(* IEC 61131-3 sources: Dev/Dev_V200/200 (part 23) *)

VAR_GLOBAL
	fb_Nh_Create_DIR		: _Nh_Create_DIR;
END_VAR

{ $DEFINE __NH_LIST_PLC_STRING }

TYPE
   NH_FRM_HED {HIDDEN}   : STRUCT      				// HLAVNA RIADIACA PREMENNA
      name     : STRING[5] :='_END';
		desc		: STRING[20];
      wht      : USINT;       	// 1-brw,2-FRM,3-MNU,4- HOME-PG - ALL, 0=read All file (log/230...)
		row		: USINT:=1;       // numbrer of Rows
		sld		: USINT;    		// number of sliders
		siz		: UDINT;				// size all file (NH_FRM_HED+data)
	END_STRUCT;

	NH_PLC_DIR_DHED       : STRUCT   	// dir
//      eTime   	: STRING[11] :='00:00:00.00'; stim 	: BYTE := 16#3b;
      dUp   	: STRING[1] :=' ';
		dEmpty	: STRING[1]	:=' ';
      dDT   	: STRING[19]:='                   ';
//		dName		: STRING;	//:='                                                                           ';
//      Cr       : BYTE   := 16#0D;
//      Lf       : BYTE   := 16#0A;
	END_STRUCT;
	{ $IFDEF __NH_LIST_PLC_STRING }
		NH_PLC_DIR_FHED       : STRUCT   // struktura EVN-log
//			aaa		: STRING[3]:= 'aaa';  s1 	: BYTE := 16#3b;
//			bbb		: STRING[3]:= 'bbb';  s2 	: BYTE := 16#3b;
   	   fLen   	: STRING[3] :='   ';
			DaysOld	: STRING[5] :='     ';
			fS			: STRING[6] :='      ';
	      fDT   	: STRING[19]:='                   ';
		END_STRUCT;
	{ $ELSE }
		NH_PLC_DIR_FHED       : STRUCT   // struktura EVN-log
   	   fLen   	: UDINT;	//STRING[3] :='   ';
			oldDays	: UINT;
			fS			: UDINT;	//STRING[10]:='          ';
	      fDT   	: DT;	//STRING[19];	//:='                   ';
		END_STRUCT;
	{ $END_IF }
	NH_PLC_DIR_DATA       : STRUCT   // struktura EVN-log
		dHed		: NH_PLC_DIR_DHED;			// DIR info
		dName		: STRING[100];	//:='                                                                           ';
		fHed		: NH_PLC_DIR_FHED;		// hed of file
		fName		: STRING[100];					// fileName
	END_STRUCT;

	NH_PLC_DIR_IO 	     : STRUCT   	// dir
		lenRow:			USINT:=100;		// line length in file dir
//		lenPath:			USINT:=100;
		fPdir:			UDINT;	 		// DIR-file position for return back
		fSdir:			UDINT;			// DIR-file size
		hDir: 			HANDLE;
		hLsD: 			HANDLE;
		hLsF: 			HANDLE;
		Info: 			TFileInfo;
		DaysOld: 		LONGTIME; 			// log text length

		lifeSize:		ARRAY[0..1,0..4] OF UDINT;	//[lifeTime, 1/2lifeTime, 1/4lifeTime, oneMonth]
 	END_STRUCT;

	NH_PLC_DIR_MASK	: STRUCT   	// exluse/include/mask dir or filre
		exclDirs				:	STRING[36]	:= 'JS/;JSN/;LOGS/;NOTIFY/;IMAGES/;FRM/;';	// DIRs in which files are not deleted (Mosaic and NachHouse templates)
		exclRootFiles		:	STRING[17]	:= '//;//WWW/;//NH2/;';								// roor DIRS where files in not deleted
		exclSufixFile		:	STRING[10]	:= '.NH2;.FRM;';										// .TXT;.XML;.XLS;.JS;.ICO;.CSS; fufix files to exclude
//		exclEmptDir			:	STRING[13]	:=	'/USR/;/SYS/;';										// list of empty DIRs that will not be deleted
	END_STRUCT;
END_TYPE

FUNCTION _Nh_Chk_Mask {HIDDEN}: BOOL		// check if the file/dir matches the mask
	VAR_INPUT
		what:		SINT;
	END_VAR
	VAR_IN_OUT
		path: 	STRING;
	END_VAR
	VAR_TEMP
		mask: 	NH_PLC_DIR_MASK;
//		wrk:		STRING[5];
	END_VAR
	_Nh_Chk_Mask := FALSE;
	CASE what OF
		1: // exlcude Suffix
			yTx0			:= MID(path,4,FIND(path,'.'));
			yTx0			:= CONCAT(yTx0,';');
			_Nh_Chk_Mask 	:= FIND(mask.exclSufixFile, yTx0) > 0 ;
		2: // no-delete dir
			yTx0				:= CONCAT(path,';');
			_Nh_Chk_Mask 	:= FIND(mask.exclDirs, yTx0) > 0 ;	// find p
		3: // sys dir mask - exlclude when chceck only SYS disk
			yTx0				:= CONCAT(path,';');
			_Nh_Chk_Mask 	:= FIND(mask.exclRootFiles, yTx0) > 0 ;
(*
		4: // dir from list found in path - Excl Empty Dir
			yTx0 := mask.exclEmptDir;
			del 	:= FIND(yTx0,';');
			WHILE del > 0 DO
				wrk := LEFT(yTx0,del-1);
				IF FIND(path,wrk)	> 0 THEN
					_Nh_Chk_Mask := TRUE;
					EXIT;
				ELSE
					yTx0	:= DELETE(yTx0,del,1);
					del 	:= FIND(yTx0,';');
				END_IF;
			END_WHILE;
*)
	ELSE _Nh_Chk_Mask := TRUE;
	END_CASE;
END_FUNCTION

VAR_GLOBAL
//	_Nh_Dir_Data	AT mObr 			{HIDDEN}: NH_PLC_DIR_DATA ;						// before yTx6
	_Nh_Dir_Data	 			: NH_PLC_DIR_DATA ;						// before yTx6
END_VAR

FUNCTION	_Nh_FIX_STRING_CRLF {HIDDEN}: BOOL	// fix end string and add spaces to lenngth
	VAR_INPUT
		lenTxt	:	INT;		// all length of string
	END_VAR
	VAR_IN_OUT
		Txt		:	STRING;	// string
	END_VAR
	_Nh_FIX_STRING_CRLF := TRUE;
	memsetEx(val := 16#20202020, length 	:= INT_TO_UDINT(lenTxt) - LEN(txt) - 1    ,
											dest 		:= VOID(txt),
											offDest	:= LEN(txt) + 1  ); // vymaze zbytok stringu medzerami
	memsetEx(val := 16#0a0d, 	length 	:= 2,
										dest 		:= VOID(txt),
										OffDest 	:= INT_TO_UDINT(lenTxt)-2 ); // + CRLF
END_FUNCTION

FUNCTION _Nh_PLC_DIR_Data_ADD {HIDDEN}: BOOL
	VAR_INPUT
		file:		BOOL;
	END_VAR
	VAR_IN_OUT
		IO:		NH_PLC_DIR_IO;
//		Name: 	STRING;
	END_VAR
	_Nh_PLC_DIR_Data_ADD	:= TRUE;	fRW := 0;
	IF file THEN
//		IF IO.DaysOld.Days >= UINT_TO_DINT(IO.LifeTime) THEN
//			IO.lifeSize[0] := IO.lifeSize[0] + info.fileSize;
//		END_IF;

		{ $IFDEF __NH_LIST_PLC_STRING }
(*
			yTx0	:= CONCAT(	DT_TO_STRINGF(IO.Info.modifyTime,'%TYYYY-MM-DD-hh:mm:ss;'),
									UDINT_TO_STRINGF(MAX(1,IO.info.fileSize / 1024),'%6d;'),
									_Nh_Dir_Data.fName
			);
			fRW	:= FileWrite(hFile:=IO.hLsF ,adrBuf:=PTR_TO_UDINT(ADR(yTx0)), size:=LEN(yTx0));
*)
			_Nh_Dir_Data.fHed.fDT		:= DT_TO_STRINGF(IO.Info.modifyTime,'%TYYYY-MM-DD-hh:mm:ss');
			_Nh_Dir_Data.fHed.fS			:= UDINT_TO_STRINGF(MAX(1,IO.info.fileSize / 1024),'%6d');
			sp									:= INT_TO_UDINT(LEN(_Nh_Dir_Data.fName)) + SIZEOF(_Nh_Dir_Data.fHed);
			_Nh_Dir_Data.fHed.fLen		:= UDINT_TO_STRINGF( sp,'%3u' );
			_Nh_Dir_Data.fHed.DaysOld	:= DINT_TO_STRINGF(IO.DaysOld.Days,'%5d');

		{ $ELSE }
			_Nh_Dir_Data.fHed.fDT		:= IO.Info.modifyTime;
			_Nh_Dir_Data.fHed.fS			:= MAX(1,IO.info.fileSize / 1024);
			_Nh_Dir_Data.fHed.fLen		:= INT_TO_UDINT(LEN(_Nh_Dir_Data.fName) + SIZEOF(_Nh_Dir_Data.fHed));
			sp									:= _Nh_Dir_Data.fHed.fLen;
		{ $END_IF }
		fRW	:= FileWrite(hFile:=IO.hLsF ,adrBuf:=PTR_TO_UDINT(ADR(_Nh_Dir_Data.fHed)), size:=sp );

	ELSIF FileSetPos( hFile := IO.hLsD, offset := IO.fSdir) THEN
		_Nh_Dir_Data.dHed.dUp 	:= ' ';													// flag for new DIR
		_Nh_Dir_Data.dHed.dDT	:= DT_TO_STRINGF(IO.Info.modifyTime,'%TYYYY-MM-DD-hh:mm:ss');
		_Nh_FIX_STRING_CRLF(txt	:=	_Nh_Dir_Data.dName, lenTxt	:= USINT_TO_INT(IO.lenRow) - SIZEOF(_Nh_Dir_Data.dHed));
		sp		:= USINT_TO_UDINT(IO.lenRow);
		fRW	:= FileWrite( hFile:=IO.hLsD ,adrBuf:=PTR_TO_UDINT(ADR(_Nh_Dir_Data.dHed)),size:=sp );
		IO.fSdir := IO.fSdir + fRW;
		IO.fPdir	:= IO.fSdir;
	ELSE
		rb	:=	_NhSysLogMsg(ini:=0, msg:=' ! Err:_Nh_Dir_Data_ADD-1; fN={'+ _Nh_Dir_Data.dName + '}; fSdir='+UDINT_TO_STRING(IO.fSdir) );
	END_IF;
	IF fRW <> sp THEN
		rb		:=	_NhSysLogMsg(ini:=0, msg:=' ! Err:_Nh_Dir_Data_ADD-2; fN={'+ _Nh_Dir_Data.dName + '}; fRW: '+UDINT_TO_STRING(fRW));
		_Nh_PLC_DIR_Data_ADD	:= FALSE;
	END_IF;
END_FUNCTION

FUNCTION_BLOCK _Nh_PLC_DIR  // list DIR and save to file in RAM
	VAR_INPUT
		Go: 				USINT; 			// 1=start list DIR, 2=next entry, 0=stop
		dirName:    	STRING[40]; // DIR path is first condition, then Case disk
		usr:     		USINT;   	// make list to user work Dir (only when GoDelete=FALSE)
		lifeTime: 		UINT:=730; 	// how many days older files will be deleted/tested
		noSubDir:		BOOL;			//	Not go to Sudirectories
		checkFile:		BOOL:=TRUE;	// first create list DIRs and check and writes files
		emptyDir:		BOOL:=TRUE;	// second check empty Dirs in list ONLY !! Empty DIRs (AND delete  IF GoDelete:=TRUE)
		// parameters Only for delete/test
		GoDelete:		BOOL:=TRUE;	// list DIRs without excludeDirs (files will remain) and net DELETE/TEST
		testOnly: 		BOOL:=TRUE; // only tests, does not delete (only when GoDelete:=TRUE)
		append:			BOOL;			// append to DEL_RRMM.log (only if )
	END_VAR
	VAR_OUTPUT
		busy: 			BOOL;
		done: 			BOOL;
		tree:				BOOL;			// 1.cycle = create DIR tree
		errID:			USINT;
		nCyc:				UINT;
	END_VAR
	VAR
		IO:				NH_PLC_DIR_IO;
	END_VAR
	VAR_TEMP
		ok1:				BOOL;
//		mask: 			NH_PLC_DIR_MASK;
	END_VAR
	done	:= FALSE;
	CASE go OF
		0: RETURN;
		1:		// start list DIR with disk
				Go	:=	10; busy	:= TRUE;	errID	:= 0; IO.fPdir	:= 0; IO.fSdir	:= 0; nCyc := 0; tree:=TRUE;
				rb := memset(val := 0, length := SIZEOF(IO.lifeSize), dest := VOID( IO.lifeSize ));
				IF GoDelete THEN usr	:= 0;	END_IF;				// system DIR
				yTx0 := MID(dirName,1,1);
				IF dirName = '' OR yTx0 <> '/' THEN
					dirName := '//';															// root
				END_IF;
				yTx0	:= MID(dirName,1,LEN(dirName));									// last char in dirName for DIR/file
				IF	yTx0 <> '/' THEN
					dirName := CONCAT(dirName,'/');										// add at the End DIR
				END_IF;
				rb := _NhSysLogMsg(msg:='->Start scan DIRs: {'+dirName+'}');
				// DIR log
				rb	:=	_Nh_Log_Path(wh:=24, frm:=3, wh2:=usr);	// yTx1	:=	'/RAM/USR/{usr}/PLC_DIR.log', if wh2:=0 '/RAM/SYS/PLC_DIR.log'
				IF _NhFdelete( fN:=yTx1, fH:=IO.hLsD, open:=TRUE, mode:=F_READ_PLUS  ) = FALSE THEN
					errID	:=	2; yTx0 	:= CONCAT('IO.hLsD:{',yTx1,'}');
				END_IF;
				// FILES log
				IF GoDelete = FALSE 	THEN	rb	:=	_Nh_Log_PATH(wh:=24, frm:=4, wh2:=usr);	// list only all files		-> PLC_FILE.log
				ELSIF testOnly 		THEN	rb	:=	_Nh_Log_PATH(wh:=24, frm:=5, wh2:=1);	// list of test-delete file 	-> TST_RRMM.log
				ELSE								rb	:=	_Nh_Log_PATH(wh:=24, frm:=5, wh2:=2);	// list of deleted filed 		-> DEL_RRMM.log
				END_IF;
				IF GoDelete AND append  THEN
					IF _NhFopen( fN:=yTx1, fH:=IO.hLsF, mode:=F_APPEND, close:=TRUE ) = FALSE THEN
						errID	:=	2; yTx0 	:= CONCAT('append: IO.hLsF:{',yTx1,'}');
					END_IF;
				ELSIF _NhFdelete( fN:=yTx1, fH:=IO.hLsF, open:=TRUE, mode:=F_APPEND  ) = FALSE THEN 	// F_READ_PLUS
					errID	:=	2; yTx0 	:= CONCAT(yTx0,'delete: IO.hLsF:{',yTx1,'}');
				END_IF;
				IF errID > 0 THEN
					yTx0 := CONCAT(' Err: ',yTx0);
				ELSE
					yTx0	:= CONCAT('DELETED files from Root: {',dirName,'}'
										,'; lifeTime: ',UINT_TO_STRING(lifeTime)
										,' ; SubDir: ',BOOL_TO_STRINGF(noSubDir,'%b{N^Y}')
										,'; EmptyDir: ',BOOL_TO_STRINGF(emptyDir,'%b{Y^N}')
										,'; checkFile: ',BOOL_TO_STRINGF(checkFile,'%b{Y^N}')
										 );
					rb	:=	_NhSysLogMsg(msg:=yTx0,openfH:=IO.hLsF, ini:=FALSE,eRowBefore:=TRUE,eRowAfter:=TRUE,maxSize:=0);
					_Nh_Dir_Data.dName		:= dirName;
					_Nh_Dir_Data.dHed.dUp := 'R';													// sign for next cycle, that DIR pased
					_Nh_PLC_DIR_Data_ADD( IO:=IO);	//, Name:=dirName );					// add 1.line to PLC_DIR.log
				END_IF;

//				IO.hDir := INVALID_HANDLE_VALUE;

		10:	// read nex file/DIR or open new DIR
				ok1	:= IO.hDir <> INVALID_HANDLE_VALUE;									// DIRs is open
				IF ok1 THEN
					ok1 := DirRead(hDir := IO.hDir, dirInfo := IO.Info);	   		// read next file/DIR
//					_Nh_Dir_Data.dHed.dUp := ' ';													// sign for next cycle, that DIR pased
					IF ok1 THEN ;																	// ADD dir/file
					ELSIF noSubDir THEN															// End of DIR, No Search in Subdir
						Go	:= 99;																	// Go previous dir
						RETURN;
					ELSE																				// End of DIR
						rb := _NhFclose(fH:=IO.hDir, dir:=TRUE);
						Go	:= 12;																	// Go previous dir
						RETURN;
					END_IF;
				END_IF;
				IF ok1 = FALSE THEN
					IO.hDir	:= DirOpen( dirName := dirName, dirinfo:=IO.Info );
					IF IO.hDir = INVALID_HANDLE_VALUE THEN
						// Empty Dir - from 12-previous DID or from 3-start
						IF IO.fPdir > 0 THEN
							IF tree=FALSE AND emptyDir THEN
								IF 	FIND(dirName,aSys.YYYY_MM) > 0 THEN;				// actual mont DIRs '2025_05/'
//								ELSIF FIND(dirName,'/SYS/') > 0 THEN;						// RAM/SYS/
								ELSIF FIND(dirName,'/USR/') > 0 THEN;						// RAM/USR/*
								ELSE
									rb	:=	_NhSysLogMsg(msg:=dirName,openfH:=IO.hLsF, ini:=FALSE,noTime:=TRUE,maxSize:=0);
//									rb	:=	_NhSysLogMsg(ini:=0, msg:=' EMPTY-Dir: {'+dirName+'} fP:'+UDINT_TO_STRING(IO.fPdir));
								END_IF;
							END_IF;
							Go	:=	12;
//							RETURN;
						ELSE
							yTx0	:=	CONCAT('  ! Err: DirOpen {',dirName,'}; fN: {',IO.Info.fileName,'}');
							errID	:=	10;
						END_IF;
					ELSIF tree = FALSE THEN
//						rb := _NhFclose(fH:=IO.hDir, dir:=TRUE);
						Go	:=	12;
//						RETURN;
					ELSE
						ok1	:=	TRUE;
					END_IF;
				END_IF
				IF ok1 THEN
					Go	:=	10;																							// next file in Dir
					yTx0 := MID(IO.Info.fileName,1,LEN(IO.Info.fileName));								// last char in dirName for check if DIR or file
					IF IO.info.fileName = '' THEN																// no file in new open DIR / unknown err
						ErrID := 10;
						yTx0 := 'IO.info.fileName=""';
					ELSIF yTx0 = '/' THEN																				// is DIR
						ok1 := TRUE;
						IF 	IO.info.fileName = 'USB/' THEN	ok1 := aSys.DiskHed.disk[2].Exist;
						ELSIF IO.info.fileName = 'SDC/' THEN	ok1 := aSys.DiskHed.disk[3].Exist;
						ELSIF IO.info.fileName = 'RAM/' THEN	ok1 := aSys.DiskHed.disk[4].Exist;
						ELSIF GoDelete = FALSE 	THEN ; 																	// list writes all files
						ELSIF _Nh_Chk_Mask(what:=2, path:=IO.info.fileName) THEN	ok1 := FALSE;
						END_IF;
						IF ok1 THEN
							_Nh_Dir_Data.dName := CONCAT(dirName,IO.Info.fileName);
							rb := _Nh_PLC_DIR_Data_ADD( IO:=IO ); 				 								// OK: add new rec with DIR
						END_IF;
//					ELSIF false	THEN		// file
					ELSIF checkFile	THEN		// file
						ok1	:=	TRUE; 								// Write
						IF 	GoDelete = FALSE 	THEN	; 												// list writes all files
						ELSIF _Nh_Chk_Mask(what:=3, path:=dirName) THEN	ok1 := FALSE;
						END_IF;
						IF ok1 THEN
							_Nh_Dir_Data.fName	:= CONCAT(dirName,IO.info.fileName,_Nh_CRLF);
							IO.DaysOld := SUB_DT_DT_LONG(aSys.NhDT, IO.Info.modifyTime);

							IF IO.DaysOld.Days >= UINT_TO_DINT(LifeTime) THEN
								IO.lifeSize[0,0] := IO.lifeSize[0,0] + 1;
								IO.lifeSize[1,0] := IO.lifeSize[1,0] + IO.info.fileSize;
							ELSIF IO.DaysOld.Days >= UINT_TO_DINT(LifeTime/2) THEN
								IO.lifeSize[0,1] := IO.lifeSize[0,1] + 1;
								IO.lifeSize[1,1] := IO.lifeSize[1,1] + IO.info.fileSize;
							ELSIF IO.DaysOld.Days >= UINT_TO_DINT(LifeTime/4) THEN
								IO.lifeSize[0,2] := IO.lifeSize[0,2] + 1;
								IO.lifeSize[1,2] := IO.lifeSize[1,2] + IO.info.fileSize;
							ELSIF IO.DaysOld.Days >= 31 THEN
								IO.lifeSize[0,3] := IO.lifeSize[0,3] + 1;
								IO.lifeSize[1,3] := IO.lifeSize[1,3] + IO.info.fileSize;
							ELSE
								IO.lifeSize[0,4] := IO.lifeSize[0,4] + 1;
								IO.lifeSize[1,4] := IO.lifeSize[1,4] + IO.info.fileSize;
							END_IF;

							_Nh_PLC_DIR_Data_ADD( IO:=IO, file:=TRUE );
						END_IF;
					END_IF;
				END_IF;

		12:	// Go Up to previous DIR
				IF IO.fPdir <= USINT_TO_UDINT(IO.lenRow) THEN										// 1.row i root = END
					IF tree THEN
						IF emptyDir THEN
							rb	:=	_NhSysLogMsg(msg:='Deleted EMPTY DIRs:',openfH:=IO.hLsF,ini:=FALSE,eRowBefore:=TRUE,eRowAfter:=TRUE,maxSize:=0);
						END_IF;
						IO.fPdir	:= IO.fSdir;
						tree		:= FALSE;																	// 2.cycle = check Empty DIRs
						Go := 12;
					ELSE
						Go	:=	99;
					END_IF;
				ELSE
					IO.fPdir	:= IO.fPdir - USINT_TO_UDINT(IO.lenRow);
					IF FileSetPos( hFile := IO.hLsD, offset := IO.fPdir) THEN					// previous (Up) Dir
						fRW	:=	FileRead(hFile:=IO.hLsD ,adrBuf:=PTR_TO_UDINT(ADR(_Nh_Dir_Data.dHed)),size:=USINT_TO_UDINT(IO.lenRow));
						dirName	:= _Nh_Dir_Data.dName;													// set Actual DIR for check file
						IF tree = FALSE THEN																	// 1.cycle = create DIR
							rb := _NhFclose(fH:=IO.hDir, dir:=TRUE);
							Go	:= 10;																			// Go next DIR (up  to file)
						ELSIF _Nh_Dir_Data.dHed.dUp <> ' ' THEN											// DIR has already been passed.
							Go	:= 12;																			// Go next DIR (up  to file)
						ELSIF FileSetPos( hFile := IO.hLsD, offset := IO.fPdir) THEN			// always=TRUE,  only to adjust begin row
							_Nh_Dir_Data.dHed.dUp := 'Y';													// sign for next cycle, that DIR pased
							fRW	:=	FileWrite( hFile:=IO.hLsD ,adrBuf:=PTR_TO_UDINT(ADR(_Nh_Dir_Data.dHed)),size:=1 );
							Go	:= 10;																			// next DIR
							IF FIND(dirName,'/.') > 0  THEN;												// Skip Hidden Dir-olny
								Go := 12;
							END_IF;
						ELSE																			// unknown Err
							errID	:=	12;
							yTx0	:=	CONCAT('Unknown Err; fP:',UDINT_TO_STRING(IO.fPdir));
						END_IF;
						rb := FileSetPos( hFile := IO.hLsD, offset := IO.fPdir);				// sets the position to the beginning of the line where DIR is loaded
					ELSE
						errID	:=	12;
						yTx0	:=	CONCAT('Err-FileSetPos(fP)=FALSE: fP:',UDINT_TO_STRING(IO.fPdir));
					END_IF;
				END_IF;

		90:	// Cancel
				errID := 90; 				// close files correctly
		99:	// END with error, OR no ERROR
				rb			:= _NhSysLogMsg(msg:='->End   scan DIRs. '+UINT_TO_STRING(nCyc)+' cyc');
				done		:=	TRUE;
				busy		:=	FALSE;
				dirName	:= '';
				rb 		:= _NhFclose(fH:=IO.hDir, dir:=TRUE);
				rb 		:= _NhFclose(fH:=IO.hLsD);
				rb 		:= _NhFclose(fH:=IO.hLsF);
				Go			:=	0;
				RETURN;
	ELSE
		errID:=100;
		yTx0	:= CONCAT('No CASE Go:=',USINT_TO_STRINGF(Go,'%3u'));
	END_CASE;
	nCyc	:= nCyc + 1;
	IF errID > 0 THEN
		Go	:=	99;
		ok1	:=	FALSE;
		ok2	:= TRUE;
		CASE errID OF
			1:		ok1	:= TRUE;		// open log-files
			10:	ok1	:= TRUE;		// open DIR
			90:	yTx0	:=	' *Cancel scan DIRs !';
		END_CASE;
		IF ok2 THEN
			yTx0	:= CONCAT(' ! Err _Nh_PLC_DIR: ',USINT_TO_STRINGF(errID,'%03u')
									,' Msg: ',yTx0
									,';hDir: ',BOOL_TO_STRINGF(IO.hDir <> INVALID_HANDLE_VALUE,'%b{Y^N}')
									,';hLsD: ',BOOL_TO_STRINGF(IO.hLsD <> INVALID_HANDLE_VALUE,'%b{Y^N}')
									,';hLsF: ',BOOL_TO_STRINGF(IO.hLsF <> INVALID_HANDLE_VALUE,'%b{Y^N}')
										);
		END_IF;
		IF ok1 THEN
				rb		:=	GetLastErrTxt(errCode:=GetLastErr(), errMessage := yTx2);
				yTx0	:= CONCAT(yTx0,';GetErr: ',yTx2);
		END_IF;
		rb := _NhSysLogMsg(msg:=yTx0);
	END_IF;
END_FUNCTION_BLOCK

VAR_GLOBAL
	fb_Nh_PLC_DIR		: _Nh_PLC_DIR;
END_VAR

FUNCTION_BLOCK _Nh_Copy_DIR // copy file or directory
	VAR_INPUT
		go: 		   USINT;			// 1=copy file, 2=copy dir and next case run
		IniEnd: 	   USINT;			// when ends set the case of main
		IniErr: 	   USINT;			// when error set the case of main
		IniRun: 	   USINT := 255;	// when start set the case of main
		copy: 		BOOL := TRUE;	// copy:=false => delete after copy (move)
		file: 		BOOL := TRUE ;	// dir or file
    	exec: 		BOOL; 			// leading edge start new write/read. if a process is running, interrupt it and close the file
		init: 		BOOL;			   // only open files an prepare for run on the next call
	END_VAR
   VAR_OUTPUT
     	done: 		BOOL; 			// action is done
     	busy: 		BOOL; 			// action in progress
     	err: 		   BOOL; 			// error flag
     	errID: 		UDINT; 			// error number
     	size: 		UDINT; 			// data length {it is entered at the beginning and cannot be changed after that !!!}
     	actSize: 	UDINT; 			// really written
		cycSize: 	UDINT; 		 	// actualy Size per cycle
		cyc: 		   UINT;			// number of cycles
		files: 		UINT;
		allSize: 	UDINT;
		_NhFileInfo: TFileInfo;
   END_VAR
   VAR
		hDir: 		HANDLE;
      hSrc: 		HANDLE;
      hDst: 		HANDLE;
      hLog: 		HANDLE;
	 	adrVar: 	   UDINT; // adresa: variable/Ram/Dbx address {it is entered at the beginning and cannot be changed after that !!!}
		GoNext: 	   USINT;
   END_VAR
	done	:= FALSE;
	CASE Go OF

     	0: RETURN;
     	1: // copy file
			// ytx3,yTx4 contain both source and destination files, including the path
			aSys.Ini	:= IniRun;
			files		:= 0;
			allSize	:= 0;
			file		:= TRUE;
			IF CPU_CODE >= 2000 THEN
				IF ForceDirs(fileName := yTx4) = FALSE THEN
					yTx2	:= yTx4;
					Go		:= 80;
					RETURN;
				END_IF;
			END_IF;
			Cyc      := 0;
         exec		:= TRUE;
			GoNext 	:=	99;                                                         // next cyccle

     	2: // Start copy DIR + first file
			// ytx3,yTx4 contain only the source and destination directories without the file
			aSys.Ini	:= IniRun;
			files		:= 0;
			allSize	:= 0;
			file		:= FALSE;                                                      // it  is DIR
			hDir		:= DirOpen(dirName := yTx3, dirInfo := _NhFileInfo);           // open DIR for read
			IF hDir = INVALID_HANDLE_VALUE THEN                                     // open error
				yTx2	:= yTx3;
				Go		:= 80;
				RETURN;
			ELSIF FileExists(fileName := yTx4) THEN	;                             // test if exist
			ELSIF CPU_CODE >= 2000 THEN
				IF ForceDirs(fileName := yTx4) = FALSE THEN
					yTx2	:= yTx4;
					Go		:= 80;
					RETURN;
				END_IF;
			ELSIF DirCreate(dirName := yTx4) 	THEN	;
			ELSE
				yTx2	:= yTx4;                                                       // create text error
				Go		:= 80;
				RETURN;
			END_IF;
			Cyc      := 0;
         exec		:= TRUE;                                                       // go directly for first file
 			GoNext	:= 12;                                                         // next cyccle

    	12: // Next file in copy DIR

			IF DirRead(hDir := hDir, dirInfo := _NhFileInfo) = FALSE THEN
				rb		:= _Nh_Log_Path(wh:=24, frm:=1, wh2:=2);																	// only log DIR {to yTx3}
				yTx2	:= CONCAT('End of dir. f:', UINT_TO_STRING(files), ' s: ', UDINT_TO_STRING(allSize) ) ;
	 		   _Nh_Line_RW(mode := 2, fH := hLog, LineLen := 0);
				Go		:= 99;
				RETURN;
			END_IF;
			exec	:= TRUE;

	 	80:	// Error
			err := TRUE;
			IF errID = 0 THEN
	 			errID := GetLastErr();
			 	GetLastErrTxt(errCode := errID, errMessage := yTx1);
				yTx2	:= CONCAT('err: ', UDINT_TO_STRING(errID), ' msg: ', yTx1, ' f: ', yTx2);
			ELSE
				yTx2	:= CONCAT('err: ', UDINT_TO_STRING(errID), ' 3: ', yTx3, ' 4: ', yTx4);
			END_IF;
			rb		:= _Nh_Log_Path(wh:=24, frm:=1, wh2:=2);															// yTx1 	:= CONCAT(aSys.ADR_RAM,'_CopyDir.log');
			_Nh_Line_RW(mode := 2, fH := hLog, LineLen := 0);
         Go    := 99;
			RETURN;

	   99:	// End
			rb		:= _NhFClose(fH := hDir, dir := TRUE);
     		IF copy = FALSE AND err = FALSE THEN								               // delete source file/dir
	 			IF file THEN                                                            // delete file
					_Nh_Line_RW(mode := 0, fH := hLog, LineNbr := 1);
   	  			IF file THEN
						yTx2	:= CONCAT('Delete file: ', yTx2) ;
					ELSE
		 				rb 	:= DirDelete(dirName := yTx2);
						yTx2	:= CONCAT('Delete dir: ', yTx2) ;
					END_IF;
					_Nh_Line_RW(mode := 2, fH := hLog, LineLen := 0);
				END_IF;
			END_IF;
     		rb 	 		:= _NhFclose(fH := hSrc);
     		rb 			:= _NhFclose(fH := hDst);
     		rb 			:= _NhFclose(fH := hLog);
			Go 			:= 0;
			GoNext 		:=	0;
			Done 		:= TRUE;
			Busy		:= FALSE;
			IF err THEN
				aSys.Ini	:= IniErr;
			ELSE
				aSys.Ini	:= IniEnd;
			END_IF;
			RETURN;

	   254: ; // TST
			   RETURN;

	   255: ; // running;

	   ELSE // non-defined
		   	aSys.Ini	:= IniRun;
			   Go 		:= 99;
			   RETURN;
   END_CASE;
   IF exec THEN
      aSys.Ini	:= IniRun;
		exec 	:= FALSE; done := TRUE; busy := FALSE; err := TRUE; errID := 0; actSize := 0;
	   IF Go < 10 THEN																	            // start copy file/Dir
			rb		:= _Nh_Log_Path(wh:=24, frm:=1, wh2:=2);															// LOG copy
   		yTx2  := yTx3;	_Nh_Line_RW(mode := 1, fH := hLog, new := TRUE, close := TRUE);
   		yTx2  := yTx4;	_Nh_Line_RW(mode := 2, fH := hLog);
		END_IF;
		IF goNext = 12 THEN
   		_Nh_Line_RW(mode := 0, fH := hLog, LineNbr := 1);	yTx3	:= CONCAT(yTx2, _NhFileInfo.fileName);
   		_Nh_Line_RW(mode := 0, fH := hLog, LineNbr := 2);	yTx4	:= CONCAT(yTx2, _NhFileInfo.fileName);
			yTx2	:= CONCAT(_NhFileInfo.fileName, ' ', UDINT_TO_STRING(_NhFileInfo.fileSize));
   		_Nh_Line_RW(mode := 2, fH := hLog, LineLen := 0);
		END_IF;
      IF _NhFopen(fN := yTx3, fH := hSrc , mode := 0) THEN 	// open source file
			size	:= FileSize(hFile := hSrc);
			IF _NhFopen(fN := yTx4, fH := hDst , mode := 1) THEN 	// open dest file
				done 		:= FALSE; busy := TRUE; err := FALSE;
				adrVar 	:= PTR_TO_UDINT( ADR(mObr) ) ;							// wrk mem used for copy
			ELSE
				errID	:= 900002;
			END_IF;
		ELSE
			errID	:= 900001;
		END_IF;
		Go 		:= 255;
		IF init THEN																		// only prepare open files/dirs
			init	:= FALSE;
			IF busy THEN
				RETURN;																		// if not Err
			END_IF;
		END_IF;
   END_IF;

   IF busy THEN
      cyc := cyc + 1;
		IF aSys.mSecMax > aSys.mSecLimit THEN
			cycSize := 512;
		ELSE
			cycSize := _NH_CLUSTER;
		END_IF;
		cycSize 	:= MIN(size - actSize, cycSize);
		fRW 		:= FileRead( hFile := hSrc, adrBuf := adrVar, size := cycSize);
		fRW 		:= FileWrite(hFile := hDst, adrBuf := adrVar, size := fRW);
     	actSize 	:= actSize + fRW; // actual read/write size
		IF actSize = size THEN
        	done := TRUE;
      ELSIF fRW <> cycSize THEN // the request did not proceed correctly
         done 	:= TRUE; err := TRUE; errID	:= 900003;
		END_IF;
	END_IF;
   IF done THEN
      rb 	   := _NhFclose(fH := hSrc);
      rb 	   := _NhFclose(fH := hDst);
		allSize	:= allSize + actSize;
		files		:= files + 1;
      IF err THEN
			GoNext	:= 80;
			files		:= 0;
		ELSIF copy = FALSE THEN
			_Nh_Line_RW(mode := 0, fH := hLog, LineNbr := 1);
			IF file = FALSE THEN
				yTx2	:= CONCAT(yTx2, _NhFileInfo.fileName);
			END_IF;
			rb 	:= FileDelete(fileName := yTx2);
      END_IF
		Go 	:= goNext;
		done	:= FALSE;
   END_IF;
END_FUNCTION_BLOCK

VAR_GLOBAL
	fb_Nh_Copy_DIR			: _Nh_Copy_DIR;
END_VAR

FUNCTION _Nh_LVL_100 {HIDDEN}: REAL // vypocita LVL 0..100 a koriguje o Minimum a Maximu
   VAR_INPUT
 		lvlIn: REAL; 	// hodnota 0..100
   	lvlMin: USINT := 10; 	// minimum 0..100
   	lvlMax: USINT := 100; // maximum 0..100
   END_VAR
   _Nh_LVL_100 := ( USINT_TO_REAL(lvlMin) + lvlIn * ( USINT_TO_REAL(lvlMax - lvlMin) / 100.0 )) * BOOL_TO_REAL(lvlIn > 0.0) ; // minimum + skorigovany LVL

// _Nh_LVL_100 := USINT_TO_REAL(lMin) + LVL*( USINT_TO_REAL(lMax-lMin)/254.0 ); // minimum + skorigovany LVL
// _Nh_LVL_100 := _Nh_LVL_100/2.54 * BOOL_TO_REAL(LVL > 0.0); // prevod na 0..100 len ked je VAL > 0
//	_Nh_LVL_100	:= ( vr + xDev^.al.ou.val * (kr - vr) / 100.0) * BOOL_TO_REAL(xDev^.al.ou.val > 0.0) ;
END_FUNCTION

FUNCTION _Nh_255_100 {HIDDEN}: REAL
   VAR_INPUT
      lvl: USINT;
   END_VAR
// _Nh_255_100 := FLOOR( USINT_TO_REAL(LVL)/2.54 );
   _Nh_255_100 := USINT_TO_REAL(LVL);
END_FUNCTION

FUNCTION_BLOCK _Nh_PWM {HIDDEN} // Blikac / Pulsne sirkova modulace
   VAR_INPUT
      Per: UINT; // perioda modulace [ms] (50-56000)
      Pls: USINT; // sirka pulsu [%] (0-100% z periody)
      Run: BOOL; // povolovaci vstup
   END_VAR
   VAR_OUTPUT
      Q: BOOL; // priznak zmeny vystupu
      Out: BOOL; // vystup
      et: UINT; // zostavajuci cas do konca periody [ms]
   END_VAR
   VAR
   END_VAR
   Q := FALSE;
   IF Run = FALSE THEN // je spusteny blikac
      et := 0;
      IF Out THEN // ak prisiel stop (run=0) v priebehu trvania impulzu, vystup mohol byt zapnuty
         Out := FALSE; // finalne vypne vystup
         Q := TRUE;
      END_IF;
   ELSIF et = 0 THEN // start
      et := MAX(50, Per);
      IF pls > 0 THEN // zapne sa len ked ma nejake trvanie
         Out := TRUE;
         Q := TRUE;
      END_IF;
   ELSE
      et := et - MIN(et, aSys.mSec);
      IF et > 0 AND Out AND pls < 100 THEN
         IF et <= REAL_TO_UINT( UINT_TO_REAL(per) * 0.01 * USINT_TO_REAL(100 - pls)) THEN // zostavanic cas je meni ako doba vypnutia (100-pls)
            Out := FALSE;
            Q := TRUE;
         END_IF;
      END_IF;
   END_IF;
END_FUNCTION_BLOCK

FUNCTION_BLOCK _Nh_Blik_FB {HIDDEN}
	VAR_INPUT
		wht: USINT;				// perioda
      nbr: USINT; // pocet zablikani
		RunOn: BOOL; // zapnut
		// future
//		RunOff: BOOL;
//		EndOn: BOOL;
//		EndOFF: BOOL;
   END_VAR
   VAR_OUTPUT
      Q: BOOL; // vystup
      Qi: BOOL; // zmena ON-OFF-ON
		Qn: BOOL; 		// imp. pri dosiahnuti poctu zaplikani
   END_VAR
   VAR
// Qr: BOOL;
      Qo: BOOL;
   END_VAR
	CASE wht OF
   	 0: Q	:= 0;
				RETURN;
		 1: Q := SYSTEM_S.PERIOD_PULSE_1SEC;					// kazdu sec
		 2: Q := SYSTEM_S.PERIOD_PULSE_10SEC;					// kazdych 10S pravidelne
		 3: IF Q THEN													// 10s je zapmute a 1s vypnute
					IF SYSTEM_S.R_EDGE_10SEC THEN
					 Q := FALSE;
					END_IF;
	 			ELSIF SYSTEM_S.R_EDGE_1SEC THEN
					Q := TRUE;
		 		END_IF;
		 5: Q := SYSTEM_S.PERIOD_PULSE_500MS;					// kazdych 500ms
		 6: Q := SYSTEM_S.PERIOD_PULSE_1MIN;					// kazdu 1.Min
				// vlastne pulzy
		100: Q := aSys.PULSE_50MS;
		101: Q := aSys.PULSE_100MS;
		102: Q := aSys.PULSE_200MS;
	END_CASE;
   Qi := Q <> Qo;
   Qo := Q;
	Qn	:= FALSE;

	IF nbr = 0 THEN
		;
	ELSIF RunON THEN
		IF	Q THEN
			RunOn 	:= FALSE;
			Qi		 	:= TRUE;
		END_IF;
	ELSIF	Qi AND Q = FALSE THEN
		nbr 	:= nbr - 1;
		IF nbr = 0 THEN
			Qn		:= TRUE;
			wht 	:= 0 ;
		END_IF;
	END_IF;
END_FUNCTION_BLOCK

FUNCTION_BLOCK _Nh_Click_FB {HIDDEN}

   VAR_OUTPUT
		Q: BOOL; // vyhodnotenie {impulz alebo ak je press alebo hold, je signal az do ukoncenia)
		Qb: BOOL;										// ak bol pri vyhodnocovani jedenehi BTN stlaceny INY BTN
		Lock: BOOL;										// WSB je zalokovane = drzi sa viac ako 10s
		Click: USINT; 	// cislo clicku na OutBTN
		OutBtn: USINT; 	// vyhodnoteny btn = InBtn pri prvom stlaceni
	END_VAR
	VAR_INPUT
		InBtn: USINT; 				// stalceny nejaky btn v sekcii CLICK ... trva asi 8 cyklov, potom 0->1
      cfc: PTR_TO NH_CFG_CLICK; 				// zaciatok CFX je rovnaky pre vsetky
		BTNs: USINT := 6;
	END_VAR
 	VAR
		trg: aTrgQx;											// vyhodnoti Qr,Q,Qf
		tClk: DT;													// strojovy cas clicku
   	Go: USINT;
		et: USINT;
	END_VAR
	Q			:= FALSE;
	Qb			:= FALSE;
	Lock		:= FALSE;
	IF trg.Qr	THEN
		IF InBtn > 0 THEN
			i			:= InBtn;
		ELSE
			FOR i := 1 TO BTNs DO
				IF xPtB^ THEN
					EXIT;
				END_IF;
				xPtB := xPtB + 1;
   		END_FOR;
		END_IF;
		IF Go = 8 THEN
			IF i <> OutBtn THEN
				xDevOkA^.al.ou.cmd	:= OutBtn;
				xDevOkA^.al.ou.par	:= USINT_TO_INT(Click);
				Qb						:= TRUE;
				Click 				:= 0;
			END_IF;
		ELSE
			Click 				:= 0;
		END_IF;
		Go 					:= 9; 										// startuje sa vzdy 1
		OutBtn				:= i;
		tClk					:= GetRTC();									// zaciatok Clicku

//		_Nh_Log_Evn_ADD( tsk := aCfg[cf].tgrp, wht := 'BEG', tRtc := tClk);

		xDevOkA^.al.ou.Val := USINT_TO_REAL(i);
		xDevOkA^.ok.ref	:= TRUE;
		xDevOkA^.al.sta	:= 1;
	ELSIF trg.Q	THEN
		_NhTime := SUB_DT_DT( GetRTC() , tClk);
		IF _NhTime > T#11s THEN
			Lock 	:= TRUE;
			Go		:= 0;
		ELSE
			CASE Go OF
   	 0: // uz sa vyhodnotil Hold, alebo aj press pred Hold, caka sa len na pustenie BTN
      	 1: // prebieha press - posielaju sa udaje pre stmievanie ....
					Q	:= TRUE;
			 2:	// bezi cakacka na Hold - kedy sa dosiahne cas;
					IF SUB_DT_DT( GetRTC() , tClk) > USINT_TO_TIME(cfc^.Hold) * 100 THEN								// HW vyhodnotil Click, mal by byt na to BTN, ktory je prve spracovavany
						Click := 7;
						Q			:= TRUE;
						Go 		:= 0;
					END_IF;
	 	ELSE
				IF _NhTime >= USINT_TO_TIME(cfc^.Press) * 100 THEN // prvykrat sa dosiahol press
					IF cfc^.Press > 0 THEN // prvykrat sa dosiahol press
						Click := 6;
						Q			:= TRUE;
					END_IF;
					IF cfc^.Hold > 0 THEN // AND cfC^.BtnHold[Btn] // kontrola, ci nie je nadefinovany Hold
      	 	Go 	:= 2;
					ELSE
						Go		:= 1;
					END_IF;
   	 END_IF;
			END_CASE;
		END_IF;
	ELSIF trg.Qf	THEN
		IF Go = 9 THEN													// prve pustenie btn
			Click := Click + 1;
			IF Click > 4 THEN										// dosakol sa MAX pocet 5-Clickov
				Q 				:= TRUE;
				Go 			:= 0;
			ELSIF cfc^.Click = 0 OR cfc^.OneClck[OutBtn] THEN	// btn NE-bude vyhodnocovat dalsi click, potvrdi sa prvy
				Q 				:= TRUE;
				Go 			:= 0;
			ELSE
				tClk	:= GetRTC();									// zaciatok Clicku
				Go 	:= 8;
         END_IF;
			et := 20;
		ELSE 													// prebieha press alebo Hold
			et := 5;
			Go 	:= 0;
		END_IF;
	ELSIF Go = 8	THEN // cakacka na dalsi click
		IF SUB_DT_DT( GetRTC() , tClk) > USINT_TO_TIME(cfc^.Click) * 100 THEN								// HW vyhodnotil Click, mal by byt na to BTN, ktory je prve spracovavany
			Q				:= TRUE;
			Go 			:= 0;
		END_IF;
	ELSIF et > 0 THEN
		IF SYSTEM_S.R_EDGE_100MS THEN
			et := et - 1;
			IF et = 0 THEN
				xDevOkA^.al.ou.val 	:= 0.0;
				xDevOkA^.ok.ref		:= TRUE;
				xDevOkA^.al.sta		:= 0;
			END_IF;
		END_IF;
	END_IF;
	IF Q THEN
		xDevOkA^.al.ou.cmd	:= OutBtn;
		xDevOkA^.al.ou.par	:= USINT_TO_INT(Click);
	ELSIF Qb = FALSE THEN
		xDevOkA^.al.ou.cmd	:= 0;
	END_IF;
END_FUNCTION_BLOCK

VAR_GLOBAL
//	fb_Nh_Copy_Dir: _Nh_Copy_Dir;

	fbFileRWa: _Nh_File_RW;
//	fbFileRWb: _Nh_File_RW;
	fbLine: _Nh_File_Line;
//	fbBrwDir: _Nh_Brw_Dir;
END_VAR

(* ---- prgMain.ST ---- *)
{ $ IFNDEF _Nh_CUST_RESTART } 	                 // ak nie je definovana funkcia v uzivatelskom subore, vytvori sa pre
(*
   FUNCTION _Nh_CUST_RESTART  {HIDDEN} : BOOL
		;
   END_FUNCTION
*)
{ $ END_IF }

TYPE _Nh_Last_State_ON : STRUCT 		// last state PRG/CPU before restart
		lastDT:		DT; (* Comment *)
		Ini: 			USINT;
		copy:		BOOL;
		cfg:		BOOL;

	END_STRUCT
END_TYPE

VAR_GLOBAL
//DeleteFiles : DeleteSurplusFilesEx := ( delEmptyDir := true ); // delete surplus files in  given  directory
  	fb_Nh_Import_CIB		: _Nh_Import_CIB;
	fb_Nh_Cfg_Restart		: _Nh_Cfg_Restart;
	fb_Nh_Log_DBX_RW		: _Nh_Log_DBX_RW;		// write log to buffer (DBx,RBx) and read from buffer and send datagram to Pi or Write to USB/LOG
END_VAR
VAR_GLOBAL RETAIN
	_NhLastPowerOffState		: _Nh_Last_State_ON; 		// last state PRG/CPU before Power OFF
END_VAR

PROGRAM prgMain
   VAR
   	fbCrHet				: _Nh_Create_HET;
      { $ IFDEF __NH_WEB }
         fbWebControl   : _NhWebControl;
      { $ END_IF  }
		ok				: BOOL;
//    	notification 	: TWebPushNotif;
//    	webPush      	: fbWebPushService;

   END_VAR
//	rb 							:= 1;
	aSys.RWtoFileCycle		:= 0;																	// how many writes to all files in cyc
	aSys.NhTime    			:= GetTime();
  	aSys.NhDate    			:= GetDate();
  	aSys.NhDT      			:= GetDateTime();													// skoro strojovy cas zaciatku cyklu, ked sa uz zapli vsetky vystupy
  	aSys.LogHed.logTime  	:= TIME_TO_STRINGF(aSys.NhTime,'%Thh:mm:ss.zz');
  	aSys.LogHed.logDate  	:= DATE_TO_STRINGF(aSys.NhDate,'%TYY-MM-DD');

	// 1   SEC 	=  10000 SYSTEM_S.LAST_CYCLE_TIME_100US      1.0 * 10 000
	// 0,7 SEC 	=  7000 SYSTEM_S.LAST_CYCLE_TIME_100US	   	0.7 * 10 000
	// 0.001    =    10
   aSys.dMin      	:= USINT_TO_INT( SYSTEM_S.COUNTER_HOURS ) * 60 + USINT_TO_INT(SYSTEM_S.COUNTER_MINUTES);  // pocet minut v ramci dna
	aSys.rSec	   	:= UINT_TO_REAL( SYSTEM_S.LAST_CYCLE_TIME_100US ) / 10.0 ;		// REAL: doba minuleho cyklu v mS (prevod zo 100 mikrosekund)
	aSys.mSec			:= REAL_TO_UINT( ROUND(  aSys.rSec ) );			            // UINT: doba minuleho cyklu v mS  (prevod zo 100 mikrosekund)
//	aSys.rTime     	:= TIME_TO_REAL(aSys.NhTime);				// REAL: cas v sekundach od polnoci

(*
	IF System_S.F_EDGE_10SEC THEN	//System_S.F_EDGE_1MIN OR  System_S.R_EDGE_1MIN THEN				// kazdych 30sec
		aSys.LogHed.Quite10Sec := aSys.LogHed.Quite10Sec + 1;
		IF aSys.LogHed.Quite10Sec > 6 THEN														// ak nebol 1 min zapis, zavrie subor
			rb := _Nh_Log_Evn_ADD(tsk := 255);
		END_IF;
		aSys.mSecMax			:= 0;
	END_IF;
*)

 	aSys.mSecMax 	:= MAX(aSys.mSec, aSys.mSecMax);
	aSys.et50		:= aSys.et50 + SYSTEM_S.LAST_CYCLE_TIME_100US;
	IF aSys.PULSE_BEEP THEN
		IF aSys.et_PULSE_BEEP > aSys.mSec THEN
			aSys.et_PULSE_BEEP := aSys.et_PULSE_BEEP - aSys.mSec;
		ELSE
			aSys.PULSE_BEEP 		:= 0;
			aSys.et_PULSE_BEEP 	:= 1000;
		END_IF;
	ELSIF asys.et_PULSE_BEEP > aSys.mSec THEN
		aSys.et_PULSE_BEEP := aSys.et_PULSE_BEEP - aSys.mSec;
	ELSE
		aSys.PULSE_BEEP		:= 1;
		aSys.et_PULSE_BEEP	:= 200;
	END_IF;

	IF aSys.et50 >= 500 THEN
		aSys.et50			:= 0;
		aSys.u50ms			:= 1;
		aSys.PULSE_50MS 	:= NOT aSys.PULSE_50MS;
	ELSE
		aSys.u50ms			:= 0;
	END_IF;
	aSys.et100		:= aSys.et100 + SYSTEM_S.LAST_CYCLE_TIME_100US;
	IF aSys.et100 >= 1000 THEN
		aSys.et100			:= 0;
		aSys.PULSE_100MS	:= NOT aSys.PULSE_100MS;
   	aSys.u100ms    	:= 1;
	ELSE
   	aSys.u100ms    := 0;
	END_IF;
	aSys.et200		:= aSys.et200 + SYSTEM_S.LAST_CYCLE_TIME_100US;
	IF aSys.et200 >= 1900 THEN
		aSys.et200			:= 0;
		aSys.PULSE_200MS 	:= NOT aSys.PULSE_200MS;
	END_IF;
	// USINT
	aSys.n1Min     := BOOL_TO_USINT(SYSTEM_S.F_EDGE_1MIN);           // kazdu 1.Min bude = 1
	aSys.n100ms    := BOOL_TO_USINT(SYSTEM_S.F_EDGE_100MS);     //;
	aSys.n50ms     := BOOL_TO_USINT(SYSTEM_S.R_EDGE_100MS OR SYSTEM_S.F_EDGE_100MS);     //;
	// UINT
	aSys.u1Min     := BOOL_TO_UINT(SYSTEM_S.F_EDGE_1MIN);           // kazdu 1.Min bude = 1
  	aSys.i1Min     := USINT_TO_INT(aSys.n1Min);           			// MIN	: INT
	// 1. sec
	IF SYSTEM_S.F_EDGE_1SEC THEN
   	aSys.n1Sec     := 1;           								// SEC	: USINT
  		aSys.u1Sec     := 1;           								// SEC	: UINT
	ELSE
   	aSys.n1Sec     := 0;
  		aSys.u1Sec     := 0;
	END_IF;
	aSys.cyc     		:= NOT aSys.Cyc;							// kazdy cyklus sa prepne
	aSys.RestCyc   	:= aSys.RestCyc + 1;

	CASE aSys.ini OF
       0:	// riadna prevadzka
			// sekvencia 3 cyklov za sebou po prechode na novu minutu, alebo natvrdo zadanim aSys.RefCycNew := true
			// 1 -> 2 -> 3 ->  0
			CASE aSys.RefCyc OF
				0:  IF aSys.RefCycNew THEN										// je zaradena nova poziadavka na restart sekvencie - zacne az ked skonci predchadzajuca sekvencia
						aSys.RefCyc		:=	1;
						aSys.RefCycNew	:= false;
					END_IF;
				3:	// obehlo 3x
					aSys.RefCyc	:=	0;
			ELSE
					aSys.RefCyc := aSys.RefCyc + 1;                 // rucne sa moze nastartovat hocikde v programe na (1), tu sa prida na (2)
			END_CASE;
(*
               Paradox( chan_code := CH5_uni, par_system_data := paradox_data,
                         max_zone_count  := paradox_max_zone_count);
               aSys.ExtPSN := Paradox.com_ok;
*)

(*)
            IF SYSTEM_S.F_EDGE_1DAY OR aSys.Restart THEN                   // novy den
					aSys.RefCyc	:=	1;														// v dalsom cykle nastartuje TypDay
	  				aMeteo.SunriseTime := SunTime( direction := Sunrise, zenith := Zenith_Official,
   		                       longitude := xGlb^.cx.longitude, latitude := xGlb^.cx.latitude,
      		                    utcOffset := UtcOffset_CR(), actDate := aSys.NhDate);
				  	aMeteo.SunsetTime := SunTime( direction := Sunset, zenith := Zenith_Official,
			   		             longitude := xGlb^.cx.longitude, latitude := xGlb^.cx.latitude,
               		          utcOffset := UtcOffset_CR(), actDate := aSys.NhDate);
					xHom^.ok.ref := true;
				ELSIF SYSTEM_S.F_EDGE_1MIN  THEN												// nastartuje 1.cyklus  - ma prednost pred vsetkym
					aSys.RefCyc	:=	1;                                  				// prvy cyklus kde sa skutocne zacne robit ma cislo  2, 3-4-5
					_NhSysUpd(fDbx:=true, file:=1);                                // Mem->RBx, ked bude file > 10 aj RBx->file
				ELSIF aSys.RefCyc	= 0 THEN
					IF aSys.RefCycNew THEN										// je zaradena nova poziadavka na restart sekvencie - zacne az ked skonci predchadzajuca sekvencia
						aSys.RefCyc		:=	1;
						aSys.RefCycNew	:= false;
					END_IF;
				ELSIF aSys.RefCyc	> 3 THEN                         	// pocita 4 cyklov za sebou od prechodu  [2..6]
					aSys.RefCyc	:=	0;
				ELSE
					aSys.RefCyc := aSys.RefCyc + 1;                 // rucne sa moze nastartovat hocikde v programe na (1), tu sa prida na (2)
				END_IF;
*)
            { $ IFDEF __NH_WEB }
               fbWebControl();
            { $ END_IF }                      // zobrazenie nastavenych DEV - za DEV. Ak sa nieco prestavi vo web v dalej otocke sa to prejavi v DEV
            { $ IFDEF __NH_WRK }
               _NhDataWrk();
			{ $ END_IF }

         _NhDevControl();           // fyzicke nastavenie DEV, malo buy byt prve
			fbNotify();
			fbWebPush();

			aSys.F_EDGE_1MIN		:= FALSE;		// vynuluje sa edge
			aSys.F_EDGE_1HOUR		:= FALSE;		// vynuluje sa edge
			aSys.F_EDGE_1DAY		:= FALSE;		// vynuluje sa edge
			aSys.F_EDGE_1MON		:= FALSE;		// vynuluje sa edge
			aSys.F_EDGE_1YEAR		:= FALSE;		// vynuluje sa edge
			aSys.Restart  			:= false;                     						// vynuluje sa restart, ale az ked sa prebehu prvykrat vsetky DEV

     	10:    ;  // nic
            rb             := _NhSysLogMsg(msg:='Check data: _Nh_DEV_RESTART');
		     	_Nh_DEV_RESTART();
            rb       		:= _NhSysLogMsg(eRowAfter:=1,msg:='*** KONIEC RESTARTU ***');
            _NhCloseAllFiles();
            aSys.ini       := 0;

		11:	// vytvori HET
				fbCrHet();
				IF aSys.ini = 0 THEN
//			      fbCrDir.go		:= -2000;
      		END_IF;

(*
     	49:    // este raz pootvarat vsetky subory
				_NhCloseAllFiles();
//				aSys.OpenFilesCount := OpenFilesCount();
      		aSys.ini    := 10;

*)
(*
            IF fbCrDir.Done THEN
               yTx2     	:= 'UKONCENE vytvaranie LOG adresarov [49]';
               rb       	:= _Nh1RowTxt(logRst:=1);
	            aSys.ini    := 10;
            END_IF;
            fbCrDir();
*)
     	40:    // Upload program
				yTx2           := CONCAT('start LoadNewPackage2:',yTx4);
            rb             := _Nh1RowTxt(logRst := 1, adTime:=3, EmpRow:=1);
				ok 				:= LoadNewPackage2( rq := true, pckg := yTx4);
            yTx2           := CONCAT('End LoadNewPackage2:',BOOL_TO_STRINGF(ok,'%b{Yes^No}' ));
            rb             := _Nh1RowTxt(logRst := 1, adTime:=3);
				aSys.ini			:= 0;

     	50:    // upravena ram do DBX
            _Nh_Go_MemToDBX();
            yTx2  := 'Na zaver upravena  RAM->DBX';
            rb             := _Nh1RowTxt(logRst := 1);
				aSys.ini       := 10;

		100:	// ulozit RAM do DBX a spustit zalohovanie dobrej DBX na SDC
            _NhWrkRam();                  // adresy WRK ram za poslednymi datami
            aSys.ini       := 50;

   	180:    // export VAZ[1..4]
				cf 		:= 1;
				nd			:= 1;
				_NhxVaz(cv:=cf,nd:=nd);
           	aSys.ini := 181;
   	181:    //
		    	IF _Nh_Vaz_LOG_CV() THEN
					cf 		:= 2;
					nd			:= 1;
					_NhxVaz(cv:=cf,nd:=nd);
	            aSys.ini       := 182;
		    	END_IF;
   	182:    //
		    	IF _Nh_Vaz_LOG_CV() THEN
					cf 		:= 3;
					nd			:= 1;
					_NhxVaz(cv:=cf,nd:=nd);
	            aSys.ini       := 183;
		    	END_IF;
   	183:    //
		    	IF _Nh_Vaz_LOG_CV() THEN
					cf 		:= 4;
					nd			:= 1;
					_NhxVaz(cv:=cf,nd:=nd);
            aSys.ini       := 184;
//	            aSys.ini       := 100;
		    	END_IF;
   	184:    //
	            aSys.ini       := 100;
		    	IF _Nh_Vaz_LOG_CV() THEN
	            aSys.ini       := 100;
		    	END_IF;

		190:    // skontroluje a prida POI
            _Nh_POI_INI();
(*
				IF _GoExp THEN
           		aSys.ini       := 180;
				ELSE
           		aSys.ini       := 100;
				END_IF;
*)

 aSys.ini := 100;

    	200:    // otestuje vazby a ich parametre
            { $IFDEF __NH_WRK }
               _NhDataWrk();
            { $END_IF }
            _NhIniVAZ();
            aSys.ini := 190;

(*
    	210:    // skontroluje konzistenciu ROM,SBJ ....., nastartuje parametre
            _Nh_Ini_DEV_Test();
           	aSys.ini       := 213;
*)

    	213:    // otestuju sa postupne vsetky CFG prida parametre k DEV
            _Nh_Ini_PAR_Test();

    	214:    // koniec testu parametrov
            aSys.ini := 200;

(*
	 	215:    // z Nh2.ADR vytvori/aktuaizuje MIESTNOSTI a DEV, alebo len aktualizuje HW-adresy
         { $IFDEF __NH_EXP }
            fb_Nh_EXP_ALL();
         { $ ELSE  }
            aSys.Ini := 210;
         { $ END_IF  }
*)

    	217:    // len pre testovanie,
// _NhIsObrOk(frm:=260);

            { $IFDEF __NH_WRK }
               _NhDataWrk();

            { $END_IF }

////***********************

    	220:    // dorobi default vety + CAT,USR,FAV,HET ...,
            _Nh_Ini_DEFAUL_CFG();    							// dorobi default data

//				aSys.ini := 217;
//RETURN;

            aSys.CfgRamOk  := true;
            _Nh_Go_MemToDBX();                           // ulozi aktualnu RAM do DBX
				aSys.ini := 222;

	 	222:    // START Import dev+HW address CIB
				yTx2 		:= 'START Import CIB';
				_Nh1RowTxt(logRst:=1); //,EmpRow:=1);
				fb_Nh_Import_CIB(Go:=1);
            { $IFDEF __NH_WRK }
               _NhDataWrk();
            { $END_IF }
				aSys.Ini 		:= 223;
	 	223:    // Running Import CIB
            fb_Nh_Import_CIB();
				IF fb_Nh_Import_CIB.err THEN
					aSys.Ini 	:= 217;
				ELSIF fb_Nh_Import_CIB.done THEN
					yTx2 	:= 'END Import CIB';
					_Nh1RowTxt(logRst:=1);
					aSys.Ini 	:= 225;
   			END_IF;

    	225:    // skontroluje konzistenciu ROM,SBJ ....., nastartuje parametre

            _Nh_Ini_DEV_Test();
				aSys.exp			:= 0;
           	aSys.ini       := 213;

    	229:    // Err section 22x
				;

(*	RESTART
	250		skontroluje DBx,RBx
				_Nh_CUST_RESTART()
	251		_Nh_Create_DIR(Go:=1)
	240-242	fb_Nh_Create_FRM	COPY NH2/200/FRM/*.* -> RAM/FRM/
	230		zisti ci mame MEM niekde zalohovanu v poradi
				1.RBx .. _NhIsDBxCfgOk(RBx:=true)
				2.File   aSys.CfgBckOk {oznaci_NhIsDBxCfgOk() }
				3.DBx	   _NhIsDBxCfgOk(), ak sa najde prekopiruje sa do RBx: DBx->RBx
	231-232	Load&Convert Old CFG->Mem (z: RBx alebo DBx)
	220		_Nh_Ini_DEFAUL_CFG() - dorobi default data
	222-223	fb_Nh_Import_CIB() :	Import dev+HW address CIB
	225		_Nh_Ini_DEV_Test()	- zakladne testy konzistencie
	213-214 	_Nh_Ini_PAR_Test();	- testy PAR + prida nove PAR
	200		_NhIniVAZ(); 			- konzistenia vazieb
	190		_Nh_POI_INI();      	- skontroluje a prida POI
	100-50	 _Nh_Go_MemToDBX(); 	- 'Na zaver upravena  RAM->DBX';
	10			_Nh_DEV_RESTART(),_NhCloseAllFiles();	- pozatvara vsetky subory na SDC a otvori _NhLangTxt
*)

	 	230:    // find CFG (aMem) in RamBox/DataBox/SDC, then copy to RamBox and then RBx->Mem
			 	IF aSys.NewDBX THEN
					aSys.CfgBckOk	:=	false;
					aSys.UseRBx	   := aSys.IS_RBx;
					rb:=_NhSysLogMsg(msg:='NEW Cfg requested !');
					aSys.Ini			:= 220;
				ELSE
					fb_Nh_Cfg_Backup.IniEnd:=230; fb_Nh_Cfg_Backup.IniErr:=239; fb_Nh_Cfg_Backup.IniRun:=255;	// predbezne
					IF aSys.IS_RBx  THEN																			// from RamBox
						IF _NhIsDBxCfgOk(RBx:=true) THEN                      						// v RBx je obraz mem
    						yTx2  		:= '->RamBOX OK.';
							aSys.UseRBx	:= true;
							aSys.Ini 	:= 231;
						ELSIF aSys.CfgBckOk THEN      															// na zaciatku je 0, potom nastavi
    						yTx2  			:= '...No-RBx,but File.Ok.{File->RBx}';
							fb_Nh_Cfg_Backup.Go		:= 12; 																		// file->RAM, next back here
						ELSIF _NhIsDBxCfgOk(RBx:=false) THEN                      					// v DBX je obraz mem
    						yTx2  		:= '..DBX-Ok.{DBX->File}';
							fb_Nh_Cfg_Backup.Go	:= 3;	   																// DBX->File
						ELSE
   	 					yTx2  			:= '...No RBx/DBx/File -> {Go empty: NewDBX=true}';
							aSys.NewDBX    := true;
						END_IF;
  					ELSIF aSys.CfgBckOk THEN																	// after
  						yTx2  := '...CPU has no RamBox,but File from DBx.Ok.{now File->Mem}';
						fb_Nh_Cfg_Backup.Go:=11; fb_Nh_Cfg_Backup.IniEnd:=220;												// file->Mem
						aSys.UseRBx	:= false;
					ELSIF _NhIsDBxCfgOk(RBx:=false) THEN                      						// v DBX je obraz mem
  						yTx2  		:= '..CPU has no RamBox,but DBX-Ok.{DBX->File}';
						fb_Nh_Cfg_Backup.Go	:= 3;	   																	// DBX->File, next back here
						aSys.UseRBx	:= true;
					ELSE
						yTx2 			:= 'CPU has no RamBox, and NOT DBX. {Go empty: NewDBX=true}';
						aSys.NewDBX := true;
					END_IF;
					rb:=_NhSysLogMsg(msg:=yTx2);
				END_IF;
//				aSys.Ini := 226;

	 	231:    // START 1.Import CFG DBX->Mem
				yTx2 		:= CONCAT('START Load & Convert Old CFG: ',BOOL_TO_STRINGF(aSys.UseRBx,'%b{Rbx^DBX}'),'->Mem.',BOOL_TO_STRINGF(xDbx^.FromDBx128,' DBx128: %b{Y^N}') );
				_Nh1RowTxt(logRst:=1); //,EmpRow:=1);
	         fb_Nh_Cfg_Restart(init:=1, wh:=0, cx:=1);
				aSys.Ini 		:= 232;

	 	232:    // Running Load Old CFG
            fb_Nh_Cfg_Restart();
				IF fb_Nh_Cfg_Restart.done THEN
					yTx2 	:= 'END Load Old CFG';
					_Nh1RowTxt(logRst:=1);
					aSys.Ini 	:= 220;
   			END_IF;

		238:    ;	//Error section 230
		239:    ;	//Error section 230
				;

	 	240:    // aktualne formulare -> NH2/200/FRM
            { $ IFDEF __NH_FRM }
					IF fb_Nh_Create_FRM.done THEN
						yTx2 		:= 'OK. New FRM';
  		 				rb 		:= _Nh1RowTxt(logRst := 1);
		            aSys.ini := 241;
					ELSIF fb_Nh_Create_FRM.busy THEN ;
					ELSE 	fb_Nh_Create_FRM(Go:=1,all:=true);
					END_IF;
					fb_Nh_Create_FRM();
            { $ ELSE }
					aSys.ini := 241;
            { $ END_IF }

		241:    // COPY NH2/200/FRM/*.* -> RAM/FRM/
            	IF aSys.DiskHed.Disk[4].Exist THEN												// RAM exist, go copy
   					_Nh_Log_Path(wh:=24, frm:=1, wh2:=1);                                  // yTx3,yTx4
	     				yTx2 		:= CONCAT('START Copy {',yTx3,'}->{',yTx4,'}');													// START Create Dir
               	rb      	:= _Nh1RowTxt(logRst := 1);
               	fb_Nh_Copy_Dir(init:=TRUE,Go:= 2,IniRun:=255,IniEnd:=242,IniErr:=249);
            	ELSE
               	aSys.Ini := 230;
            	END_IF;
	 	242:    // End Copy
				yTx2		:= CONCAT('END   Copy  f: ',UINT_TO_STRING(fb_Nh_Copy_Dir.files),' s: ',UDINT_TO_STRING(fb_Nh_Copy_Dir.allSize) )  ;
    			rb			:= _Nh1RowTxt(logRst := 1);
      		aSys.Ini := 230;
	 	249: 	// Err Copy Dir
				;
	 	250: 	// restart
  				//          aSys.prgChange    		:= PROGRAMISCHANGED();
				rb:=_NhCloseAllFiles();
				IF CPU_CODE >= 2000 THEN
					rb 					:= ResizeRamBox( newSize := 16*1024);   	// 16MB*1024 = 16384 kByte
					aSys.Size_RBx 		:= UINT_TO_UDINT( SizeOfRamBox() ) * 1024;   							// 128 kb   (128*1024=131072 Byte)
					aSys.IS_RBx			:= aSys.Size_RBx >= 16777216;
				ELSE
					aSys.IS_RBx			:= false;
					aSys.Size_RBx 		:= 0;
//					yTx1					:= 'WWW/LOGS/';
			  	END_IF;
//				yTx1		:= 'WWW/NH2/';
//				rb:=DirCreate( dirName := yTx1 );																	// create default LOG adr
				aSys.Restart     		:= TRUE;
				aSys.RefCyc				:=	1;
//				aSys.rst.In				:= true;
				aSys.CfgBckOk			:=	FALSE;																	// flag, that BckFile no-Exiat
				aSys.Size_DBx 			:= UINT_TO_UDINT( SizeOfDataBox()) * 1024;   								// 128 kb   (128*1024=131072 Byte)
				aSys.IS_DBX				:= aSys.Size_DBx >= 131072;

//				aSys.DiskHed.USB_Ready.In	:= SYSTEM_S.USB_DISK_READY;									// vynuluje sa flag USB ready
//				aSys.DiskHed.USB_Ready.Q	:= SYSTEM_S.USB_DISK_READY;									// vynuluje sa flag USB ready

				aDbx.aCfx[0]   := _cfg0;
		   	aDbx.aCfx[1]   := _par0;
	   		aDbx.aCfx[2]   := _vaz0;
		   	aDbx.vRam   	:= _Ram0;                                                         // volna ram
	      	_NheRAM();                                                                    // vymaze virtualnu RAM od vRam (za CFG/PAR/VAZ...
		   	FOR i := 2  TO _Nh_Cfg DO                                                     // offset default Empty vety
    				aCfg[i].ofs   := aCfg[i-1].ofs + aCfg[i-1].siz;
	   		END_FOR;
     			FOR i := 2  TO _Nh_Par DO                                                     // offset default Empty vety
     				aPar[i].ofs   := aPar[i-1].ofs + aPar[i-1].siz ;
     			END_FOR;
				RandomU(seed := _NhSeed, init:=true);

//				rb	:= SetValueToRamBox(ramBoxAddress:=0, length:=_NH_RAM, value := 0);

//				_Nh_CUST_RESTART();                          											// nejake vlasne veci po restarte

				IF IS_COLD_RESTART_PLC 		THEN	yTx0:='COLD';
				ELSIF IS_HOT_RESTART_PLC   THEN  yTx0:='HOT';
				ELSIF IS_RESTART_PLC       THEN  yTx0:='RST';
				ELSE 						      	   yTx0:='UNKNOWN';
				END_IF;

				SYSTEM_S.F_EDGE_1DAY 	:= true;												// simulate new day for refresh day in room/het
            aSys.Ini 					:= 251;

    	251: 	// 2.cyc After restart - create dir OK

				rb:=_NhSysLogMsg(write:=0,eRowBefore:=1,msg:=' *** '+yTx0+' RESTART ***   DBx: '+UINT_TO_STRING(SizeOfDataBox())+' kB, RBx: '+UINT_TO_STRING( SizeOfRamBox() )+BOOL_TO_STRINGF(SYSTEM_S.USB_DISK_READY, ' kB; USB:%b{Y^N}')+'   *** ');				rb:=_NhSysLogMsg(eRowAfter:=1,NoTime:=1,msg:=DT_TO_STRINGF(_NhLastPowerOffState.LastDt, '%TYY.MM.DD-hh:mm:ss.zzz ') +',Ini:='+USINT_TO_STRING(_NhLastPowerOffState.ini) );
//				_Nh_Log_Dbx_ADD(ev:='AL1',src:='PIR',key:='Pir-1',val:='On',subj:=1,rom:=101);
            aSys.Ini 				:= 241;

//            aSys.Ini 				:= 255;

	 	252:    // test
            ;
		254:    // Error
            ;
		255:    // running more like one cycle, block all function except fb_ ....
            ;
	END_CASE;

	// time events - change progtam date
	IF SYSTEM_S.F_EDGE_1DAY  THEN				   											// novy den
		aSys.F_EDGE_1DAY	:= true;														// NH event
		aSys.F_EDGE_1MON 	:= aSys.MONTH 	<> SYSTEM_S.COUNTER_MONTHS;												// NH event
		aSys.F_EDGE_1YEAR	:= aSys.YEAR 	<> SYSTEM_S.COUNTER_YEARS;
		aSys.YEAR 			:= SYSTEM_S.COUNTER_YEARS;								// Nh month
		aSys.MONTH 			:= SYSTEM_S.COUNTER_MONTHS;							//	Nh month
		aSys.DAY				:= SYSTEM_S.COUNTER_DAYS_OF_MONTH;					// Nh month
		aSys.RefCycNew		:= true;														// v dalsom cykle nastartuje TypDay
		aSys.YYYY_MM		:= CONCAT(USINT_TO_STRINGF(aSys.YEAR, '20%02d'),'_',USINT_TO_STRINGF(aSys.MONTH, '%02d'),'/');
		fb_Nh_Create_DIR.exec	:= aSys.F_EDGE_1MON ;							// vytvori nove adresare pre novy mesiac
	ELSIF  SYSTEM_S.F_EDGE_1MIN  THEN                   									// new min
		aSys.F_EDGE_1MIN			:= true;												// NH event
		aSys.F_EDGE_1HOUR			:= SYSTEM_S.F_EDGE_1MIN;						// NH event
		aSys.RefCycNew				:= true;												// v dalsom cykle nastartuje TypDay
		// after xxx seconds of error-free operation, make a CFG backup
	ELSIF aSys.RestartBck = false THEN										// este nebol urobeny backup po restarte
		IF  aSys.ini = 0 AND SYSTEM_S.COUNTER_1SEC > 4 THEN     						// 1min after restart, create backup file
			IF _NhSysUpd(fFile:=true) THEN												// Mem->RBx, ked bude file > 10 aj RBx->file
				aSys.RestartBck 	:= true;
			END_IF;
		END_IF
	END_IF;

	fb_Nh_Create_DIR();												// test and create directories
	fb_Nh_Cfg_Backup();      	// save from mRam[] to file, or restore to mRam[] from file
	fb_Nh_Copy_Dir();
//	fb_Nh_Log_DBX_RW();		// write log to buffer (DBx,RBx) and read from buffer and send datagram to Pi or Write to USB/LOG
//	fb_Nh_PLC_DIR();

	_NhLastPowerOffState.LastDt	:= aSys.NhDT;
	_NhLastPowerOffState.ini 	:= aSys.ini;
//	_NhLastStateON.ini 		:= aSys.ini;

END_PROGRAM
